% RSLogix 500 project Fail-Safe Motion Interlock System.RSS, saved by version 8.30.00.16 %
PROJECT "UNTITLED"    % processor: Bul.1763 MicroLogix 1100 Series B %

PROGRAM FILES
  LAD 2 "MAIN"  10 rungs
  LAD 3 "DIGITAL IO"  9 rungs
  LAD 4 "ANALOG IO"  2 rungs

DATA FILES
  O0 OUTPUT  7 elements
  I1 INPUT  13 elements
  S2 STATUS  66 elements
  B3 BINARY  1 elements
  T4 TIMER  1 elements
  C5 COUNTER  1 elements
  R6 CONTROL  1 elements
  N7 INTEGER  1 elements
  F8 FLOAT  1 elements

LADDER 2 "MAIN"
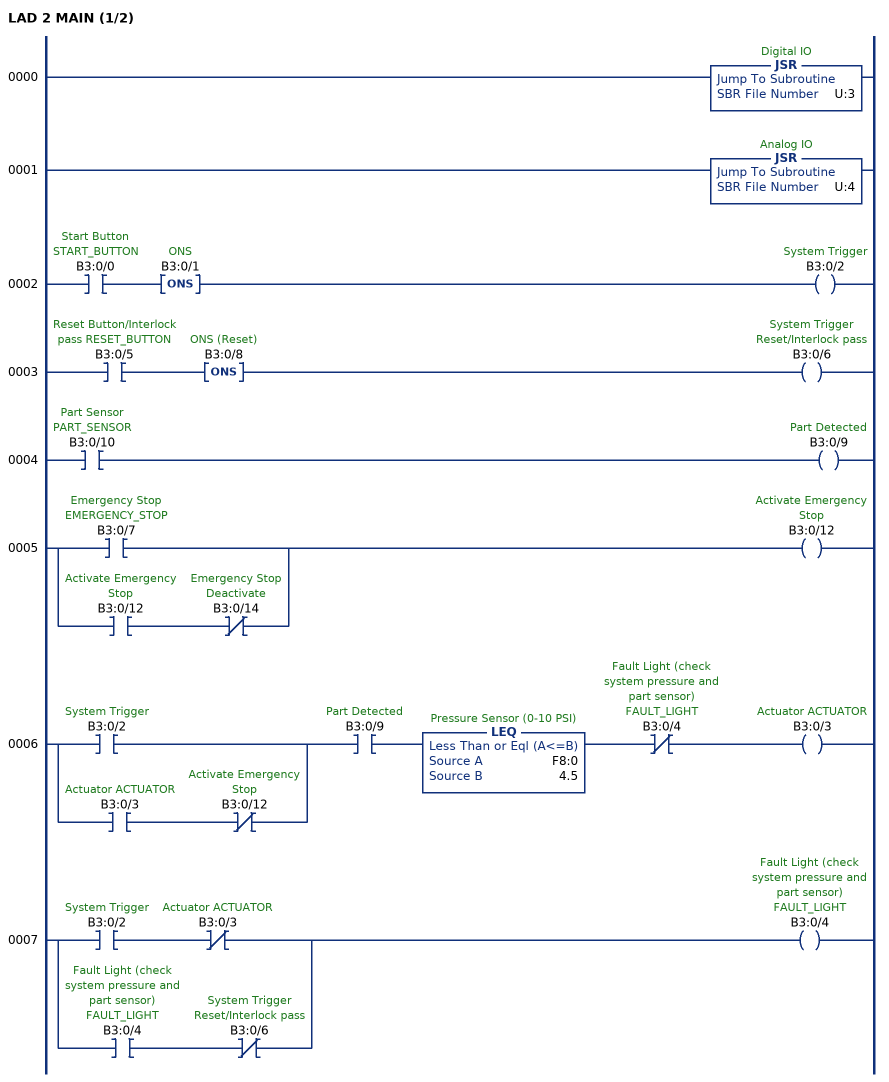
% Rung: 0 %
SOR JSR U:3 EOR
%   U:3  "Digital IO" %
% Rung: 1 %
SOR JSR U:4 EOR
%   U:4  "Analog IO" %
% Rung: 2 %
SOR XIC B3:0/0 ONS B3:0/1 OTE B3:0/2 EOR
%   B3:0/0  START_BUTTON  "Start Button" %
%   B3:0/1  "ONS" %
%   B3:0/2  "System Trigger" %
% Rung: 3 %
SOR XIC B3:0/5 ONS B3:0/8 OTE B3:0/6 EOR
%   B3:0/5  RESET_BUTTON  "Reset Button/Interlock pass" %
%   B3:0/8  "ONS (Reset)" %
%   B3:0/6  "System Trigger Reset/Interlock pass" %
% Rung: 4 %
SOR XIC B3:0/10 OTE B3:0/9 EOR
%   B3:0/10  PART_SENSOR  "Part Sensor" %
%   B3:0/9  "Part Detected" %
% Rung: 5 %
SOR BST XIC B3:0/7 NXB XIC B3:0/12 XIO B3:0/14 BND OTE B3:0/12 EOR
%   B3:0/7  EMERGENCY_STOP  "Emergency Stop" %
%   B3:0/12  "Activate Emergency Stop" %
%   B3:0/14  "Emergency Stop Deactivate" %
% Rung: 6 %
SOR BST XIC B3:0/2 NXB XIC B3:0/3 XIO B3:0/12 BND XIC B3:0/9 LEQ F8:0 4.5 XIO B3:0/4 OTE B3:0/3 EOR
%   B3:0/2  "System Trigger" %
%   B3:0/3  ACTUATOR  "Actuator" %
%   B3:0/12  "Activate Emergency Stop" %
%   B3:0/9  "Part Detected" %
%   F8:0  "Pressure Sensor (0-10 PSI)" %
%   B3:0/4  FAULT_LIGHT  "Fault Light (check system pressure and part sensor)" %
% Rung: 7 %
SOR BST XIC B3:0/2 XIO B3:0/3 NXB XIC B3:0/4 XIO B3:0/6 BND OTE B3:0/4 EOR
%   B3:0/2  "System Trigger" %
%   B3:0/3  ACTUATOR  "Actuator" %
%   B3:0/4  FAULT_LIGHT  "Fault Light (check system pressure and part sensor)" %
%   B3:0/6  "System Trigger Reset/Interlock pass" %

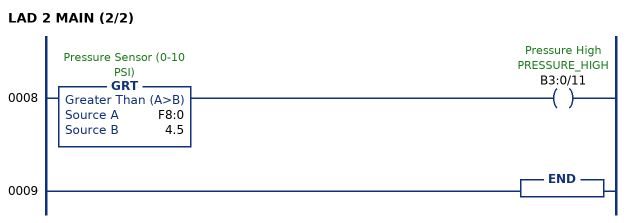
% Rung: 8 %
SOR GRT F8:0 4.5 OTE B3:0/11 EOR
%   F8:0  "Pressure Sensor (0-10 PSI)" %
%   B3:0/11  PRESSURE_HIGH  "Pressure High" %
% Rung: 9 %
SOR END EOR

LADDER 3 "DIGITAL IO"
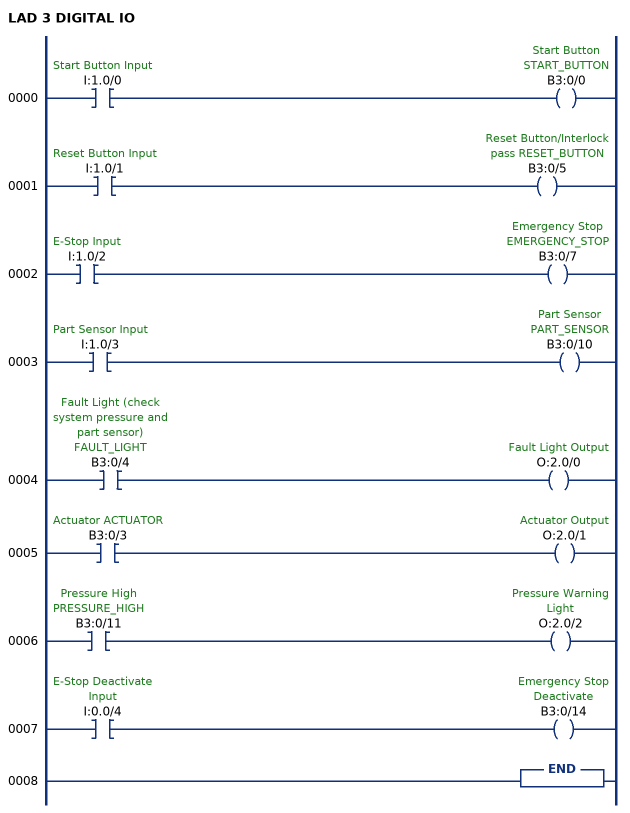
% Rung: 0 %
SOR XIC I:1.0/0 OTE B3:0/0 EOR
%   I:1.0/0  "Start Button Input" %
%   B3:0/0  START_BUTTON  "Start Button" %
% Rung: 1 %
SOR XIC I:1.0/1 OTE B3:0/5 EOR
%   I:1.0/1  "Reset Button Input" %
%   B3:0/5  RESET_BUTTON  "Reset Button/Interlock pass" %
% Rung: 2 %
SOR XIC I:1.0/2 OTE B3:0/7 EOR
%   I:1.0/2  "E-Stop Input" %
%   B3:0/7  EMERGENCY_STOP  "Emergency Stop" %
% Rung: 3 %
SOR XIC I:1.0/3 OTE B3:0/10 EOR
%   I:1.0/3  "Part Sensor Input" %
%   B3:0/10  PART_SENSOR  "Part Sensor" %
% Rung: 4 %
SOR XIC B3:0/4 OTE O:2.0/0 EOR
%   B3:0/4  FAULT_LIGHT  "Fault Light (check system pressure and part sensor)" %
%   O:2.0/0  "Fault Light Output" %
% Rung: 5 %
SOR XIC B3:0/3 OTE O:2.0/1 EOR
%   B3:0/3  ACTUATOR  "Actuator" %
%   O:2.0/1  "Actuator Output" %
% Rung: 6 %
SOR XIC B3:0/11 OTE O:2.0/2 EOR
%   B3:0/11  PRESSURE_HIGH  "Pressure High" %
%   O:2.0/2  "Pressure Warning Light" %
% Rung: 7 %
SOR XIC I:0.0/4 OTE B3:0/14 EOR
%   I:0.0/4  "E-Stop Deactivate Input" %
%   B3:0/14  "Emergency Stop Deactivate" %
% Rung: 8 %
SOR END EOR

LADDER 4 "ANALOG IO"
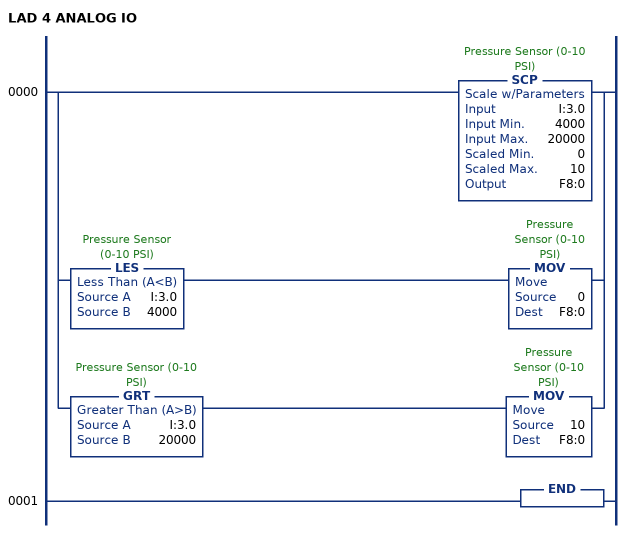
% Rung: 0 %
SOR BST SCP I:3.0 4000 20000 0 10 F8:0 NXB LES I:3.0 4000 MOV 0 F8:0 NXB GRT I:3.0 20000 MOV 10 F8:0 BND EOR
%   I:3.0  "Pressure Sensor (0-10 PSI)" %
%   F8:0  "Pressure Sensor (0-10 PSI)" %
% Rung: 1 %
SOR END EOR

OTHER DOCUMENTED ADDRESSES
  B3:0/13  "ONS (E-Stop)"
  I:3.0/0  "Pressure Sensor (0-5 PSI)"
